
// ===== library: MasterCopy "g120_init" =====

FUNCTION_BLOCK "g120_init"   // FB1, LAD
{ S7_Optimized_Access := 'TRUE' }
VERSION : 0.1
   VAR_INPUT
      start : Bool;
      direction : Bool;
      ack_error : Bool;
      Speed : UInt;
   END_VAR
   VAR_OUTPUT
      error : Bool;
      enable : Bool;
      ready : Bool;
   END_VAR
   VAR_IN_OUT
      QW_Reg : Word;
      QSpeed_Reg : UInt;
      IW_Reg : UInt;
   END_VAR
BEGIN

REGION Network 1: Set Buffer
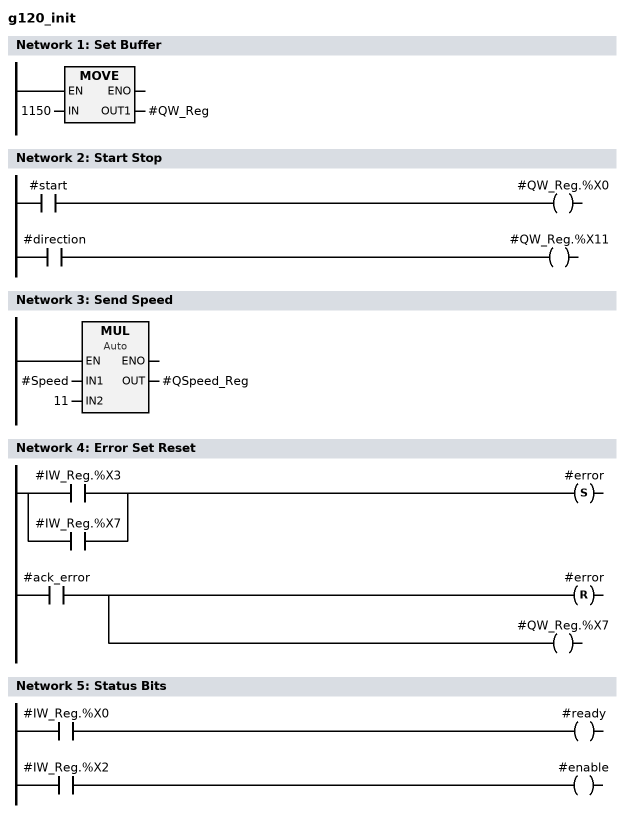
   RUNG wire#powerrail
      Move(in := 1150, out1 => #QW_Reg)
   END_RUNG
   // the same network as SCL:
   #QW_Reg := 1150;
END_REGION

REGION Network 2: Start Stop
   RUNG wire#powerrail
      Contact( #start )
      Coil( #QW_Reg.%X0 )
   END_RUNG
   RUNG wire#powerrail
      Contact( #direction )
      Coil( #QW_Reg.%X11 )
   END_RUNG
   // the same network as SCL:
   #QW_Reg.%X0 := #start;
   #QW_Reg.%X11 := #direction;
END_REGION

REGION Network 3: Send Speed
   RUNG wire#powerrail
      Mul(in1 := #Speed, in2 := 11, out => #QSpeed_Reg)
   END_RUNG
   // the same network as SCL:
   #QSpeed_Reg := #Speed * 11;
END_REGION

REGION Network 4: Error Set Reset
   RUNG wire#powerrail
      Contact( #IW_Reg.%X3 )
      wire#w1
      S_Coil( #error )
   END_RUNG
   RUNG wire#powerrail
      Contact( #IW_Reg.%X7 )
   END_RUNG wire#w1
   RUNG wire#powerrail
      Contact( #ack_error )
      wire#w2
      R_Coil( #error )
   END_RUNG
   RUNG wire#w2
      Coil( #QW_Reg.%X7 )
   END_RUNG
   // the same network as SCL:
   IF #IW_Reg.%X3 OR #IW_Reg.%X7 THEN #error := TRUE; END_IF;
   IF #ack_error THEN #error := FALSE; END_IF;
   #QW_Reg.%X7 := #ack_error;
END_REGION

REGION Network 5: Status Bits
   RUNG wire#powerrail
      Contact( #IW_Reg.%X0 )
      Coil( #ready )
   END_RUNG
   RUNG wire#powerrail
      Contact( #IW_Reg.%X2 )
      Coil( #enable )
   END_RUNG
   // the same network as SCL:
   #ready := #IW_Reg.%X0;
   #enable := #IW_Reg.%X2;
END_REGION
END_FUNCTION_BLOCK

// ===== library: MasterCopy "g120_init_v2" =====

FUNCTION_BLOCK "g120_init"   // FB1, LAD
{ S7_Optimized_Access := 'TRUE' }
VERSION : 0.1
// commissioning biterken hız referansı gireleceği zaman 16384 yazar isek gönderdiğimiz hız birebir olur.
   VAR_INPUT
      start : Bool;
      direction : Bool;
      ack_error : Bool;
      Speed : UInt;
   END_VAR
   VAR_OUTPUT
      error : Bool;
      enable : Bool;
      ready : Bool;
   END_VAR
   VAR_IN_OUT
      QW_Reg : Word;
      QSpeed_Reg : UInt;
      IW_Reg : UInt;
   END_VAR
BEGIN

REGION Network 1: Set Buffer
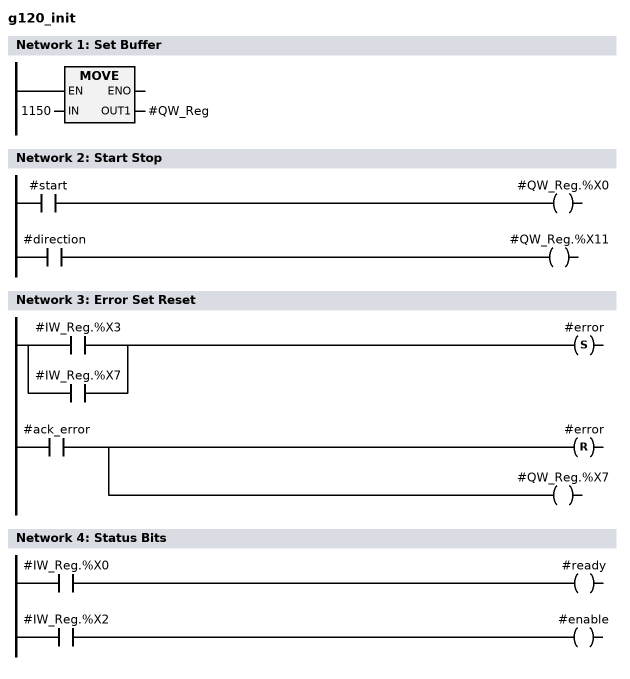
   RUNG wire#powerrail
      Move(in := 1150, out1 => #QW_Reg)
   END_RUNG
   // the same network as SCL:
   #QW_Reg := 1150;
END_REGION

REGION Network 2: Start Stop
   RUNG wire#powerrail
      Contact( #start )
      Coil( #QW_Reg.%X0 )
   END_RUNG
   RUNG wire#powerrail
      Contact( #direction )
      Coil( #QW_Reg.%X11 )
   END_RUNG
   // the same network as SCL:
   #QW_Reg.%X0 := #start;
   #QW_Reg.%X11 := #direction;
END_REGION

REGION Network 3: Error Set Reset
   RUNG wire#powerrail
      Contact( #IW_Reg.%X3 )
      wire#w1
      S_Coil( #error )
   END_RUNG
   RUNG wire#powerrail
      Contact( #IW_Reg.%X7 )
   END_RUNG wire#w1
   RUNG wire#powerrail
      Contact( #ack_error )
      wire#w2
      R_Coil( #error )
   END_RUNG
   RUNG wire#w2
      Coil( #QW_Reg.%X7 )
   END_RUNG
   // the same network as SCL:
   IF #IW_Reg.%X3 OR #IW_Reg.%X7 THEN #error := TRUE; END_IF;
   IF #ack_error THEN #error := FALSE; END_IF;
   #QW_Reg.%X7 := #ack_error;
END_REGION

REGION Network 4: Status Bits
   RUNG wire#powerrail
      Contact( #IW_Reg.%X0 )
      Coil( #ready )
   END_RUNG
   RUNG wire#powerrail
      Contact( #IW_Reg.%X2 )
      Coil( #enable )
   END_RUNG
   // the same network as SCL:
   #ready := #IW_Reg.%X0;
   #enable := #IW_Reg.%X2;
END_REGION
END_FUNCTION_BLOCK

// ===== library: MasterCopy "g120_init_v3" =====

FUNCTION_BLOCK "g120_init"   // FB1, LAD
{ S7_Optimized_Access := 'TRUE' }
VERSION : 0.1
// commissioning biterken hız referansı gireleceği zaman 16384 yazar isek gönderdiğimiz hız birebir olur.
   VAR_INPUT
      start : Bool;
      direction : Bool;
      ack_error : Bool;
      Speed : UInt;
      "first initialize" : Bool;
   END_VAR
   VAR_OUTPUT
      error : Bool;
      enable : Bool;
      ready : Bool;
   END_VAR
   VAR_IN_OUT
      QW_Reg : Word;
      QSpeed_Reg : UInt;
      IW_Reg : UInt;
   END_VAR
BEGIN

REGION Network 1: Set Buffer
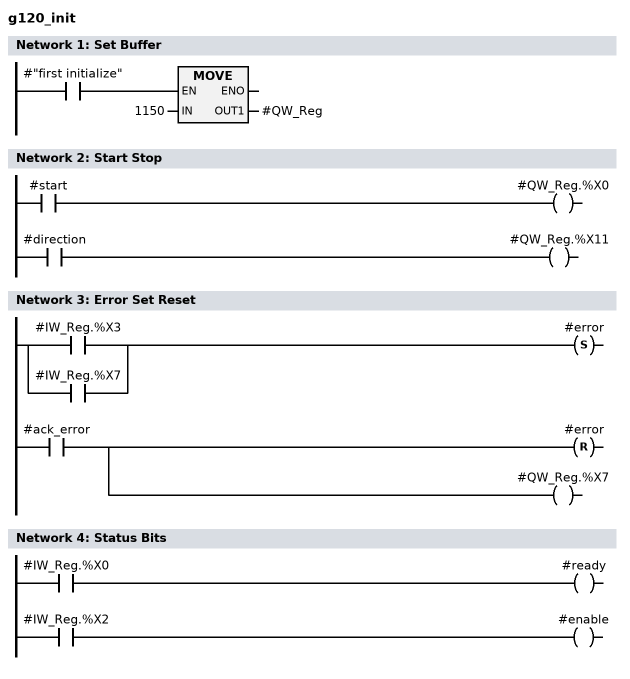
   RUNG wire#powerrail
      Contact( #"first initialize" )
      Move(in := 1150, out1 => #QW_Reg)
   END_RUNG
   // the same network as SCL:
   IF #"first initialize" THEN #QW_Reg := 1150; END_IF;
END_REGION

REGION Network 2: Start Stop
   RUNG wire#powerrail
      Contact( #start )
      Coil( #QW_Reg.%X0 )
   END_RUNG
   RUNG wire#powerrail
      Contact( #direction )
      Coil( #QW_Reg.%X11 )
   END_RUNG
   // the same network as SCL:
   #QW_Reg.%X0 := #start;
   #QW_Reg.%X11 := #direction;
END_REGION

REGION Network 3: Error Set Reset
   RUNG wire#powerrail
      Contact( #IW_Reg.%X3 )
      wire#w1
      S_Coil( #error )
   END_RUNG
   RUNG wire#powerrail
      Contact( #IW_Reg.%X7 )
   END_RUNG wire#w1
   RUNG wire#powerrail
      Contact( #ack_error )
      wire#w2
      R_Coil( #error )
   END_RUNG
   RUNG wire#w2
      Coil( #QW_Reg.%X7 )
   END_RUNG
   // the same network as SCL:
   IF #IW_Reg.%X3 OR #IW_Reg.%X7 THEN #error := TRUE; END_IF;
   IF #ack_error THEN #error := FALSE; END_IF;
   #QW_Reg.%X7 := #ack_error;
END_REGION

REGION Network 4: Status Bits
   RUNG wire#powerrail
      Contact( #IW_Reg.%X0 )
      Coil( #ready )
   END_RUNG
   RUNG wire#powerrail
      Contact( #IW_Reg.%X2 )
      Coil( #enable )
   END_RUNG
   // the same network as SCL:
   #ready := #IW_Reg.%X0;
   #enable := #IW_Reg.%X2;
END_REGION
END_FUNCTION_BLOCK